PROGRAM Recorder
VAR
	bRunning 	: BOOL;
	bGetValues 	: BOOL; //Signal from HMI that we want to read the saved values.
	//bRecord5axis : BOOL;
	
	

	nArrayIndex : INT;
	nEntryCount : INT; //How many entries exist for HMI to fetch.
	aPositions	: ARRAY[0..2048] OF LREAL;
	aCopy		: ARRAY[0..2048] OF LREAL; //HMI will fetch from aCopy and we can continue filling aPositions with new data.
	
	nIter		: INT;
	nIterMax 	: INT;
	
	//We don't know what motors the user will or will not have.
	//So IGEMS CNC sets these pointers to the adress of the motor position it wants to record.
	pAdresses : ARRAY[0..5] OF POINTER TO LREAL;
END_VAR

IF bGetValues	THEN 
	nEntryCount := nArrayIndex;
	nArrayIndex := 0;
	
	MEMCPY(destAddr:= ADR(aCopy), srcAddr:= ADR(aPositions), n:= INT_TO_UDINT(8 * nEntryCount)); 
	bGetValues := FALSE;
END_IF


IF NOT bRunning THEN
	nArrayIndex := 0;
	RETURN;
END_IF



IF (nArrayIndex > 2048) THEN
	nArrayIndex := 0; //Wrapover if no one fetched the stored values.
END_IF

(*
IF(bRecord5axis) THEN
	nIterMax := 4;
ELSE
	nIterMax := 1;
END_IF
*)


FOR nIter := 0 TO nIterMax DO
	//Get the act pos value.
	IF (pAdresses[nIter] <> 0) THEN 
		aPositions[nArrayIndex] := pAdresses[nIter]^; //Valid pointer has been set by over ADS, dereference it.
	ELSE 
		aPositions[nArrayIndex] := 0.0; //Not a valid pointer, just set the actual postion to 0.0
	END_IF
	
	nArrayIndex := nArrayIndex + 1;  
END_FOR;

END_PROGRAM

(* stored: Version 1.1.0.1, ProductVersion 3.1.4024.12
   POU Recorder: Id {fdb4ad7d-6ad0-4333-b3fc-1fe457939e3a}, SpecialFunc None *)
